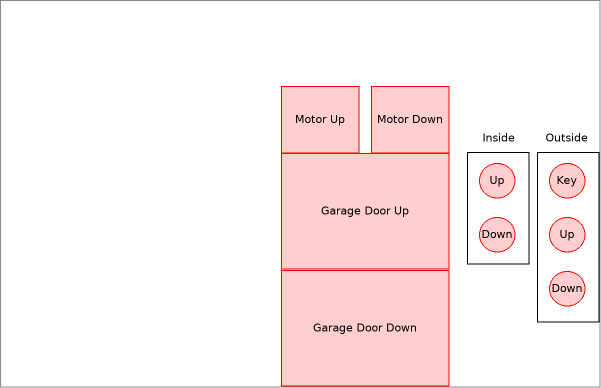
VISUALIZATION Visualization  // 601x388
    Rectangle (281,86 78x67), "Motor Up", colour toggle: POU.motor_up
    Rectangle (467,152 62x112)
    Rectangle (537,152 62x170)
    Ellipse (479,163 36x35), "Up", colour toggle: POU.up_inside
        OnMouseDown: toggle POU.up_inside
    Ellipse (549,163 36x35), "Key", colour toggle: POU.key
        OnMouseDown: toggle POU.key
    Ellipse (549,217 36x35), "Up", colour toggle: POU.up_outside
        OnMouseDown: toggle POU.up_outside
    Ellipse (549,271 36x35), "Down", colour toggle: POU.down_outside
        OnMouseDown: toggle POU.down_outside
    Ellipse (479,217 36x35), "Down", colour toggle: POU.down_inside
        OnMouseDown: toggle POU.down_inside
    Rectangle (281,153 168x116), "Garage Door Up", colour toggle: POU.door_up
        OnMouseDown: toggle POU.door_up
        OnMouseDown: toggle POU.door_up
    Rectangle (371,86 78x67), "Motor Down", colour toggle: POU.motor_down
    Rectangle (281,270 168x116), "Garage Door Down", colour toggle: POU.door_down
        OnMouseDown: toggle POU.door_down
    Label (474,123 50x30), "Inside"
    Label (542,123 50x30), "Outside"
END_VISUALIZATION

(* stored: Version 1.1.0.1, ProductVersion 3.1.4022.7
   Visu Visualization: Id {7fbe7916-74a4-4b01-8862-c0eed6f76f4d} *)
